FUNCTION_BLOCK FB_TopElement1 EXTENDS FB_BaseTopElement IMPLEMENTS ITF_TopElement1, ITF_TopElement1_HMI_Init
VAR
	itfGE1				: ITF_GroupE_TE1;

	itfCE1				: ITF_ControlE_TE1;
	itfCE2				: ITF_ControlE_TE1;

	itfC1				: ITF_Component_TE1;
	itfC2				: ITF_Component_TE1;
	itfC3				: ITF_Component_TE1;
END_VAR

METHOD FB_init : BOOL
VAR_INPUT
	bInitRetains : BOOL; // if TRUE, the retain variables are initialized (warm start / cold start)
	bInCopyCode : BOOL;  // if TRUE, the instance afterwards gets moved into the copy code (online change)
	itfGE1				: ITF_GroupE_TE1;
	itfCE1				: ITF_ControlE_TE1;
	itfCE2				: ITF_ControlE_TE1;
	itfC1				: ITF_Component_TE1;
	itfC2				: ITF_Component_TE1;
	itfC3				: ITF_Component_TE1;
END_VAR
THIS^.itfGE1 := itfGE1;
THIS^.SetText (eLocation := E_BaseLocation.pl, wsDescription := "Element złożony 1");
THIS^.SetText (eLocation := E_BaseLocation.en, wsDescription := "Element złożony 1");
THIS^.SetText (eLocation := E_BaseLocation.de, wsDescription := "Element złożony 1");
itfGE1.SetName (stName := THIS^.GetTexts ());
THIS^.AddControlElement (itfControlElement := itfGE1);

THIS^.itfCE1 := itfCE1;
THIS^.SetText (eLocation := E_BaseLocation.pl, wsDescription := "Element wykonawczy 1");
THIS^.SetText (eLocation := E_BaseLocation.en, wsDescription := "Element wykonawczy 1");
THIS^.SetText (eLocation := E_BaseLocation.de, wsDescription := "Element wykonawczy 1");
itfCE1.SetName (stName := THIS^.GetTexts ());
THIS^.AddControlElement (itfControlElement := itfCE1);

THIS^.itfCE2 := itfCE2;
THIS^.SetText (eLocation := E_BaseLocation.pl, wsDescription := "Element wykonawczy 2");
THIS^.SetText (eLocation := E_BaseLocation.en, wsDescription := "Element wykonawczy 2");
THIS^.SetText (eLocation := E_BaseLocation.de, wsDescription := "Element wykonawczy 2");
itfCE2.SetName (stName := THIS^.GetTexts ());
THIS^.AddControlElement (itfControlElement := itfCE2);


THIS^.itfC1 := itfC1;
THIS^.SetText (eLocation := E_BaseLocation.pl, wsDescription := "Komponent 1");
THIS^.SetText (eLocation := E_BaseLocation.en, wsDescription := "Komponent 1");
THIS^.SetText (eLocation := E_BaseLocation.de, wsDescription := "Komponent 1");
itfC1.SetName (stName := THIS^.GetTexts ());
THIS^.AddComponent (itfComponent := itfC1);

THIS^.itfC2 := itfC2;
THIS^.SetText (eLocation := E_BaseLocation.pl, wsDescription := "Komponent 2");
THIS^.SetText (eLocation := E_BaseLocation.en, wsDescription := "Komponent 2");
THIS^.SetText (eLocation := E_BaseLocation.de, wsDescription := "Komponent 2");
itfC2.SetName (stName := THIS^.GetTexts ());
THIS^.AddComponent (itfComponent := itfC2);

THIS^.itfC3 := itfC3;
THIS^.SetText (eLocation := E_BaseLocation.pl, wsDescription := "Komponent 3");
THIS^.SetText (eLocation := E_BaseLocation.en, wsDescription := "Komponent 3");
THIS^.SetText (eLocation := E_BaseLocation.de, wsDescription := "Komponent 3");
itfC3.SetName (stName := THIS^.GetTexts ());
THIS^.AddComponent (itfComponent := itfC3);
END_METHOD

END_FUNCTION_BLOCK

(* stored: Version 1.1.0.1, ProductVersion 3.1.4024.15
   POU FB_TopElement1: Id {bd8dcea8-d375-471b-8272-e0cf58be6ef6}, SpecialFunc None
   Method FB_init: Id {101c9f0e-95f4-4048-85ab-daec86aba431} *)
